# EPICS IOC start-up script: examples/test/PSI/ep2308.iocsh
#- mXsXXX naming
require ecmccfg, "NAMING=mXsXXX"

#- add slaves
${SCRIPTEXEC} ${ecmccfg_DIR}addSlave.cmd, "HW_DESC=EP2308, SLAVE_ID=${SLAVE=5}"
